FUNCTION_BLOCK FB_MockAxis EXTENDS SPT_Components.FB_Component_BasicAxis
VAR
    _MockInPosition : BOOL := TRUE;
    _MockBusy       : BOOL := FALSE;
	_Enabled		: BOOL := FALSE;
END_VAR

PROPERTY Busy : BOOL
GET
Busy := _MockBusy;
END_GET
END_PROPERTY

METHOD Enable : BOOL
_Enabled := TRUE;
Enable := TRUE;
END_METHOD

PROPERTY Enabled : BOOL
GET
Enabled := _Enabled;
END_GET
END_PROPERTY

PROPERTY InPosition : BOOL
GET
InPosition := _MockInPosition;
END_GET
END_PROPERTY

METHOD MoveAbsolute : BOOL
VAR_INPUT
	Position	  : LREAL;
	AbortPrevious : BOOL;
END_VAR
_MockBusy := FALSE;
_MockInPosition := TRUE;
END_METHOD

END_FUNCTION_BLOCK

(* stored: Version 1.1.0.1, ProductVersion 3.1.4024.15
   POU FB_MockAxis: Id {f3603fea-aa28-47ef-b114-9fa5d52e454a}, SpecialFunc None
   Property Busy: Id {25ee96b4-f935-48d1-85b2-42045a8b8f79}
   Get Get: Id {2073e439-15b7-4d8e-a4dd-8977881cdaca}
   Method Enable: Id {9481627a-d7cd-4736-ba69-511ff810e00c}
   Property Enabled: Id {f38a9161-cb22-4c87-a85a-6e4ede124720}
   Get Get: Id {8455ef28-d601-480d-94b2-053ea389c0b8}
   Property InPosition: Id {899ba792-f147-4840-9190-c11ac913d37c}
   Get Get: Id {f5f86ed6-a8c0-44cb-80db-e88896583828}
   Method MoveAbsolute: Id {ce2fcb65-7db9-4fdb-91ae-b88cee0c9fe3} *)
